// 画像取込可能な状態にする　【ライブ表示状態（常時連続取込）/ハードウェアトリガー版】
FUNCTION Vision_StartAcquiring_ExTrigger : ETcVnCameraState
VAR_INPUT
	fbCamera				: FB_VN_SimpleCameraControl;	// Cameraオブジェクト or File Sourceオブジェクト
END_VAR

VAR
	hr						: HRESULT;						// 関数の戻り値を表す変数
	eState					: ETcVnCameraState;				// オブジェクトの状態を表す
END_VAR

// カメラのステータスを取得
eState := fbCamera.GetState();

IF eState = TCVN_CS_ERROR THEN
	// エラーの時はリセットを実行
	hr := fbCamera.Reset();
	
ELSIF eState < TCVN_CS_ACQUIRING THEN
	// 取込開始状態に移行させる
	hr := fbCamera.StartAcquisition();
END_IF

Vision_StartAcquiring_ExTrigger := eState;

END_FUNCTION

(* stored: Version 1.1.0.1, ProductVersion 3.1.4024.12
   POU Vision_StartAcquiring_ExTrigger: Id {f462b106-1bed-4708-b1c4-56a72d3cb301}, SpecialFunc None *)
